// TIA Portal V19 export
DATA_BLOCK "PPrgArchive11"   // DB502
// stored: IsOnlyStoredInLoadMemory true, MemoryReserve 0, Namespace G
   VAR RETAIN
      PRG : Array[1001..1100] of "PPrg_Data";
   END_VAR
BEGIN
END_DATA_BLOCK
